# EPICS substitutions: ek9000App/Db/EL2808_mbboDirect.substitutions
file EL2808.template
{       pattern
        {
                TERMINAL,

        }
        {
        }
}
